# EPICS substitutions: iocBoot/iocThorLabs/AptDC.substitutions
file "$(TOP)/db/motor.db"
{
pattern
{P,         M,              DTYP,       PORT,       ADDR,   DESC,                   EGU,    DIR,    VELO,   VBAS,   ACCS,   ACCL,   BDST,   BVEL,   BACC,   MRES,               PREC,   DHLM,   DLLM,   TWV,    INIT}
#{Motor:,    "DC1",          "asynMotor","APT-DC1",  0,      "KDC101 DC Servo",      mm,     Pos,    2.3,    0.1,    1.5,    0,      2.3,    1.0,    0.000028939405515,  4,      25.0,   -0.1,   1.0,    ""}
{Motor:,    "KIM101_1",      "asynMotor",   "APT-KIM101",  0,    "Thorlabs PIA13",    steps,     Pos,    500,    100,    1000,    1,      0,    500, 1000,   1,  0,      1000000.0,   -1000000, 250,    ""}
{Motor:,    "KIM101_2",      "asynMotor",   "APT-KIM101",  1,    "Thorlabs PIA13",    steps,     Pos,    500,    100,    1000,    1,      0,    500, 1000,   1,  0,      1000000.0,   -1000000, 250,    ""}
{Motor:,    "KIM101_3",      "asynMotor",   "APT-KIM101",  2,    "Thorlabs PIA13",    steps,     Pos,    500,    100,    1000,    1,      0,    500, 1000,   1,  0,      1000000.0,   -1000000, 250,    ""}
{Motor:,    "KIM101_4",      "asynMotor",   "APT-KIM101",  3,    "Thorlabs PIA13",    steps,     Pos,    500,    100,    1000,    1,      0,    500, 1000,   1,  0,      1000000.0,   -1000000, 250,    ""}
}
